PROGRAM ProcessLamp
VAR
END_VAR

// Written 10.08.2023 by Daniel Kelly

// The purpose of this POU is to provide control to the lamps on the 
// front of the cabinet via their switches

drive.bM1active := drive.bM1switch;
drive.bM2active := drive.bM2switch; 
drive.bProcessActive := drive.bShortFeed OR drive.bStartProcess;
drive.bRemovalSequenceLamp := drive.RemovalSwitch;
drive.bValveLamp := drive.ValveSwitch;

END_PROGRAM

(* stored: Version 1.1.0.1, ProductVersion 3.1.4024.12
   POU ProcessLamp: Id {747cf198-3ab4-4dbe-86f1-8743c6f4571b}, SpecialFunc None *)
